(* IEC 61131-3 sources: TA/Tests/Diagnostic/Unitbus 0 (32) (part 2) *)

(* ---- UB_local_0_36_AIG16.st ---- *)
PROGRAM UB_local_0_36_AIG16

(***************************************************************************)
// НАСТРОЙКА ФБ
(***************************************************************************)

UB_0_32_AIG16_CH0_VAL_QUALITY_AD.Valid_down := AD_VALID_DOWN;
UB_0_32_AIG16_CH0_VAL_QUALITY_AD.Valid_up := AD_VALID_UP;
UB_0_32_AIG16_CH0_VAL_QUALITY_AD.IN0 := AD_IN0;
UB_0_32_AIG16_CH0_VAL_QUALITY_AD.IN100 := AD_IN100;

UB_0_32_AIG16_CH4_VAL_QUALITY_AD.Valid_down := AD_VALID_DOWN;
UB_0_32_AIG16_CH4_VAL_QUALITY_AD.Valid_up := AD_VALID_UP;
UB_0_32_AIG16_CH4_VAL_QUALITY_AD.IN0 := AD_IN0;
UB_0_32_AIG16_CH4_VAL_QUALITY_AD.IN100 := AD_IN100;

UB_0_32_AIG16_CH8_VAL_QUALITY_AD.Valid_down := AD_VALID_DOWN;
UB_0_32_AIG16_CH8_VAL_QUALITY_AD.Valid_up := AD_VALID_UP;
UB_0_32_AIG16_CH8_VAL_QUALITY_AD.IN0 := AD_IN0;
UB_0_32_AIG16_CH8_VAL_QUALITY_AD.IN100 := AD_IN100;

UB_0_32_AIG16_CH12_VAL_QUALITY_AD.Valid_down := AD_VALID_DOWN;
UB_0_32_AIG16_CH12_VAL_QUALITY_AD.Valid_up := AD_VALID_UP;
UB_0_32_AIG16_CH12_VAL_QUALITY_AD.IN0 := AD_IN0;
UB_0_32_AIG16_CH12_VAL_QUALITY_AD.IN100 := AD_IN100;

(***************************************************************************)
// СБРОС ОШИБОК
(***************************************************************************)

IF UB_0_32_AIG16_KVIT
    THEN UB_0_32_AIG16_KVIT := FALSE;
END_IF;

(***************************************************************************)
// КАНАЛ 0
(***************************************************************************)

UB_0_32_AIG16_CH0_VAL_MEASUREMENT := _IO_I21_AIG16_0_VAL.Measurement;

//Отказ сигнала
IF INT14(ANY_TO_DINT(_IO_I21_AIG16_0_VAL.Quality))
    THEN UB_0_32_AIG16_CH0_VAL_QUALITY_FAULT := TRUE;
    ELSE UB_0_32_AIG16_CH0_VAL_QUALITY_FAULT := FALSE;
END_IF;

// Проверка на ошибку
IF _IO_I21_AIG16_0_VAL.Quality = 0
    THEN UB_0_32_AIG16_CH0_VAL_QUALITY_ERROR := TRUE;
    ELSE UB_0_32_AIG16_CH0_VAL_QUALITY_ERROR := FALSE;
END_IF;

(***************************************************************************)
// КАНАЛ 4
(***************************************************************************)

UB_0_32_AIG16_CH4_VAL_MEASUREMENT := _IO_I21_AIG16_4_VAL.Measurement;

//Отказ сигнала
IF INT14(ANY_TO_DINT(_IO_I21_AIG16_4_VAL.Quality))
    THEN UB_0_32_AIG16_CH4_VAL_QUALITY_FAULT := TRUE;
    ELSE UB_0_32_AIG16_CH4_VAL_QUALITY_FAULT := FALSE;
END_IF;

// Проверка на ошибку
IF _IO_I21_AIG16_4_VAL.Quality = 0
    THEN UB_0_32_AIG16_CH4_VAL_QUALITY_ERROR := TRUE;
    ELSE UB_0_32_AIG16_CH4_VAL_QUALITY_ERROR := FALSE;
END_IF;

(***************************************************************************)
// КАНАЛ 8
(***************************************************************************)

UB_0_32_AIG16_CH8_VAL_MEASUREMENT := _IO_I21_AIG16_8_VAL.Measurement;

//Отказ сигнала
IF INT14(ANY_TO_DINT(_IO_I21_AIG16_8_VAL.Quality))
    THEN UB_0_32_AIG16_CH8_VAL_QUALITY_FAULT := TRUE;
    ELSE UB_0_32_AIG16_CH8_VAL_QUALITY_FAULT := FALSE;
END_IF;

// Проверка на ошибку
IF _IO_I21_AIG16_8_VAL.Quality = 0
    THEN UB_0_32_AIG16_CH8_VAL_QUALITY_ERROR := TRUE;
    ELSE UB_0_32_AIG16_CH8_VAL_QUALITY_ERROR := FALSE;
END_IF;

(***************************************************************************)
// КАНАЛ 12
(***************************************************************************)

UB_0_32_AIG16_CH12_VAL_MEASUREMENT := _IO_I21_AIG16_12_VAL.Measurement;

//Отказ сигнала
IF INT14(ANY_TO_DINT(_IO_I21_AIG16_12_VAL.Quality))
    THEN UB_0_32_AIG16_CH12_VAL_QUALITY_FAULT := TRUE;
    ELSE UB_0_32_AIG16_CH12_VAL_QUALITY_FAULT := FALSE;
END_IF;

// Проверка на ошибку
IF _IO_I21_AIG16_12_VAL.Quality = 0
    THEN UB_0_32_AIG16_CH12_VAL_QUALITY_ERROR := TRUE;
    ELSE UB_0_32_AIG16_CH12_VAL_QUALITY_ERROR := FALSE;
END_IF;

(***************************************************************************)
// ИНТЕГРАЛЬНЫЕ ПОКАЗАТЕЛИ
(***************************************************************************)

// Интегральный показателшь VAL.Quality
IF NOT INT0(UB_0_32_AIG16_CH0_VAL_QUALITY) AND
    NOT INT0(UB_0_32_AIG16_CH4_VAL_QUALITY) AND
    NOT INT0(UB_0_32_AIG16_CH8_VAL_QUALITY) AND
    NOT INT0(UB_0_32_AIG16_CH12_VAL_QUALITY)

    THEN UB_0_32_AIG16_INTEGRAL_VAL_QUALITY := TRUE;
    ELSE UB_0_32_AIG16_INTEGRAL_VAL_QUALITY := FALSE;
END_IF;

(***************************************************************************)
// ДИАГНОСТИКА ШИНЫ
(***************************************************************************)

// Диагностика 1 группы
// Адресное пространство не было найдено в Ubusdb
IF
    // Канал 0
    NOT INT4(ANY_TO_DINT(_IO_I21_AIG16_0_VAL.Quality)) AND
    NOT INT5(ANY_TO_DINT(_IO_I21_AIG16_0_VAL.Quality)) AND
    NOT INT6(ANY_TO_DINT(_IO_I21_AIG16_0_VAL.Quality)) AND
    NOT INT7(ANY_TO_DINT(_IO_I21_AIG16_0_VAL.Quality)) AND

    // Канал 1
    NOT INT4(ANY_TO_DINT(_IO_I21_AIG16_1_VAL.Quality)) AND
    NOT INT5(ANY_TO_DINT(_IO_I21_AIG16_1_VAL.Quality)) AND
    NOT INT6(ANY_TO_DINT(_IO_I21_AIG16_1_VAL.Quality)) AND
    NOT INT7(ANY_TO_DINT(_IO_I21_AIG16_1_VAL.Quality)) AND

    // Канал 2
    NOT INT4(ANY_TO_DINT(_IO_I21_AIG16_2_VAL.Quality)) AND
    NOT INT5(ANY_TO_DINT(_IO_I21_AIG16_2_VAL.Quality)) AND
    NOT INT6(ANY_TO_DINT(_IO_I21_AIG16_2_VAL.Quality)) AND
    NOT INT7(ANY_TO_DINT(_IO_I21_AIG16_2_VAL.Quality)) AND

    // Канал 3
    NOT INT4(ANY_TO_DINT(_IO_I21_AIG16_3_VAL.Quality)) AND
    NOT INT5(ANY_TO_DINT(_IO_I21_AIG16_3_VAL.Quality)) AND
    NOT INT6(ANY_TO_DINT(_IO_I21_AIG16_3_VAL.Quality)) AND
    NOT INT7(ANY_TO_DINT(_IO_I21_AIG16_3_VAL.Quality))

    THEN UB_0_32_AIG16_UNITBUS_VAL_QUALITY_GROUP_1 := 0;
END_IF;

// Не сошлась контрольная сумма данных
IF
    // Канал 0
    INT4(ANY_TO_DINT(_IO_I21_AIG16_0_VAL.Quality)) AND
    NOT INT5(ANY_TO_DINT(_IO_I21_AIG16_0_VAL.Quality)) AND
    NOT INT6(ANY_TO_DINT(_IO_I21_AIG16_0_VAL.Quality)) AND
    NOT INT7(ANY_TO_DINT(_IO_I21_AIG16_0_VAL.Quality)) AND

    // Канал 1
    INT4(ANY_TO_DINT(_IO_I21_AIG16_1_VAL.Quality)) AND
    NOT INT5(ANY_TO_DINT(_IO_I21_AIG16_1_VAL.Quality)) AND
    NOT INT6(ANY_TO_DINT(_IO_I21_AIG16_1_VAL.Quality)) AND
    NOT INT7(ANY_TO_DINT(_IO_I21_AIG16_1_VAL.Quality)) AND

    // Канал 2
    INT4(ANY_TO_DINT(_IO_I21_AIG16_2_VAL.Quality)) AND
    NOT INT5(ANY_TO_DINT(_IO_I21_AIG16_2_VAL.Quality)) AND
    NOT INT6(ANY_TO_DINT(_IO_I21_AIG16_2_VAL.Quality)) AND
    NOT INT7(ANY_TO_DINT(_IO_I21_AIG16_2_VAL.Quality)) AND

    // Канал 3
    INT4(ANY_TO_DINT(_IO_I21_AIG16_3_VAL.Quality)) AND
    NOT INT5(ANY_TO_DINT(_IO_I21_AIG16_3_VAL.Quality)) AND
    NOT INT6(ANY_TO_DINT(_IO_I21_AIG16_3_VAL.Quality)) AND
    NOT INT7(ANY_TO_DINT(_IO_I21_AIG16_3_VAL.Quality))

    THEN UB_0_32_AIG16_UNITBUS_VAL_QUALITY_GROUP_1 := 1;
END_IF;

// Не выставлены биты достоверности элементов в АП
IF
    // Канал 0
    NOT INT4(ANY_TO_DINT(_IO_I21_AIG16_0_VAL.Quality)) AND
    INT5(ANY_TO_DINT(_IO_I21_AIG16_0_VAL.Quality)) AND
    NOT INT6(ANY_TO_DINT(_IO_I21_AIG16_0_VAL.Quality)) AND
    NOT INT7(ANY_TO_DINT(_IO_I21_AIG16_0_VAL.Quality)) AND

    // Канал 1
    NOT INT4(ANY_TO_DINT(_IO_I21_AIG16_1_VAL.Quality)) AND
    INT5(ANY_TO_DINT(_IO_I21_AIG16_1_VAL.Quality)) AND
    NOT INT6(ANY_TO_DINT(_IO_I21_AIG16_1_VAL.Quality)) AND
    NOT INT7(ANY_TO_DINT(_IO_I21_AIG16_1_VAL.Quality)) AND

    // Канал 2
    NOT INT4(ANY_TO_DINT(_IO_I21_AIG16_2_VAL.Quality)) AND
    INT5(ANY_TO_DINT(_IO_I21_AIG16_2_VAL.Quality)) AND
    NOT INT6(ANY_TO_DINT(_IO_I21_AIG16_2_VAL.Quality)) AND
    NOT INT7(ANY_TO_DINT(_IO_I21_AIG16_2_VAL.Quality)) AND

    // Канал 3
    NOT INT4(ANY_TO_DINT(_IO_I21_AIG16_3_VAL.Quality)) AND
    INT5(ANY_TO_DINT(_IO_I21_AIG16_3_VAL.Quality)) AND
    NOT INT6(ANY_TO_DINT(_IO_I21_AIG16_3_VAL.Quality)) AND
    NOT INT7(ANY_TO_DINT(_IO_I21_AIG16_3_VAL.Quality))

    THEN UB_0_32_AIG16_UNITBUS_VAL_QUALITY_GROUP_1 := 2;
END_IF;

// Полученные данные корректны
IF
    // Канал 0
    INT4(ANY_TO_DINT(_IO_I21_AIG16_0_VAL.Quality)) AND
    INT5(ANY_TO_DINT(_IO_I21_AIG16_0_VAL.Quality)) AND
    NOT INT6(ANY_TO_DINT(_IO_I21_AIG16_0_VAL.Quality)) AND
    NOT INT7(ANY_TO_DINT(_IO_I21_AIG16_0_VAL.Quality)) AND

    // Канал 1
    INT4(ANY_TO_DINT(_IO_I21_AIG16_1_VAL.Quality)) AND
    INT5(ANY_TO_DINT(_IO_I21_AIG16_1_VAL.Quality)) AND
    NOT INT6(ANY_TO_DINT(_IO_I21_AIG16_1_VAL.Quality)) AND
    NOT INT7(ANY_TO_DINT(_IO_I21_AIG16_1_VAL.Quality)) AND

    // Канал 2
    INT4(ANY_TO_DINT(_IO_I21_AIG16_2_VAL.Quality)) AND
    INT5(ANY_TO_DINT(_IO_I21_AIG16_2_VAL.Quality)) AND
    NOT INT6(ANY_TO_DINT(_IO_I21_AIG16_2_VAL.Quality)) AND
    NOT INT7(ANY_TO_DINT(_IO_I21_AIG16_2_VAL.Quality)) AND

    // Канал 3
    INT4(ANY_TO_DINT(_IO_I21_AIG16_3_VAL.Quality)) AND
    INT5(ANY_TO_DINT(_IO_I21_AIG16_3_VAL.Quality)) AND
    NOT INT6(ANY_TO_DINT(_IO_I21_AIG16_3_VAL.Quality)) AND
    NOT INT7(ANY_TO_DINT(_IO_I21_AIG16_3_VAL.Quality))

    THEN UB_0_32_AIG16_UNITBUS_VAL_QUALITY_GROUP_1 := 3;
END_IF;

// Диагностика 2 группы
// Адресное пространство не было найдено в Ubusdb
IF
    // Канал 4
    NOT INT4(ANY_TO_DINT(_IO_I21_AIG16_4_VAL.Quality)) AND
    NOT INT5(ANY_TO_DINT(_IO_I21_AIG16_4_VAL.Quality)) AND
    NOT INT6(ANY_TO_DINT(_IO_I21_AIG16_4_VAL.Quality)) AND
    NOT INT7(ANY_TO_DINT(_IO_I21_AIG16_4_VAL.Quality)) AND

    // Канал 5
    NOT INT4(ANY_TO_DINT(_IO_I21_AIG16_5_VAL.Quality)) AND
    NOT INT5(ANY_TO_DINT(_IO_I21_AIG16_5_VAL.Quality)) AND
    NOT INT6(ANY_TO_DINT(_IO_I21_AIG16_5_VAL.Quality)) AND
    NOT INT7(ANY_TO_DINT(_IO_I21_AIG16_5_VAL.Quality)) AND

    // Канал 6
    NOT INT4(ANY_TO_DINT(_IO_I21_AIG16_6_VAL.Quality)) AND
    NOT INT5(ANY_TO_DINT(_IO_I21_AIG16_6_VAL.Quality)) AND
    NOT INT6(ANY_TO_DINT(_IO_I21_AIG16_6_VAL.Quality)) AND
    NOT INT7(ANY_TO_DINT(_IO_I21_AIG16_6_VAL.Quality)) AND

    // Канал 7
    NOT INT4(ANY_TO_DINT(_IO_I21_AIG16_7_VAL.Quality)) AND
    NOT INT5(ANY_TO_DINT(_IO_I21_AIG16_7_VAL.Quality)) AND
    NOT INT6(ANY_TO_DINT(_IO_I21_AIG16_7_VAL.Quality)) AND
    NOT INT7(ANY_TO_DINT(_IO_I21_AIG16_7_VAL.Quality))

    THEN UB_0_32_AIG16_UNITBUS_VAL_QUALITY_GROUP_2 := 0;
END_IF;

// Не сошлась контрольная сумма данных
IF
    // Канал 4
    INT4(ANY_TO_DINT(_IO_I21_AIG16_4_VAL.Quality)) AND
    NOT INT5(ANY_TO_DINT(_IO_I21_AIG16_4_VAL.Quality)) AND
    NOT INT6(ANY_TO_DINT(_IO_I21_AIG16_4_VAL.Quality)) AND
    NOT INT7(ANY_TO_DINT(_IO_I21_AIG16_4_VAL.Quality)) AND

    // Канал 5
    INT4(ANY_TO_DINT(_IO_I21_AIG16_5_VAL.Quality)) AND
    NOT INT5(ANY_TO_DINT(_IO_I21_AIG16_5_VAL.Quality)) AND
    NOT INT6(ANY_TO_DINT(_IO_I21_AIG16_5_VAL.Quality)) AND
    NOT INT7(ANY_TO_DINT(_IO_I21_AIG16_5_VAL.Quality)) AND

    // Канал 6
    INT4(ANY_TO_DINT(_IO_I21_AIG16_6_VAL.Quality)) AND
    NOT INT5(ANY_TO_DINT(_IO_I21_AIG16_6_VAL.Quality)) AND
    NOT INT6(ANY_TO_DINT(_IO_I21_AIG16_6_VAL.Quality)) AND
    NOT INT7(ANY_TO_DINT(_IO_I21_AIG16_6_VAL.Quality)) AND

    // Канал 7
    INT4(ANY_TO_DINT(_IO_I21_AIG16_7_VAL.Quality)) AND
    NOT INT5(ANY_TO_DINT(_IO_I21_AIG16_7_VAL.Quality)) AND
    NOT INT6(ANY_TO_DINT(_IO_I21_AIG16_7_VAL.Quality)) AND
    NOT INT7(ANY_TO_DINT(_IO_I21_AIG16_7_VAL.Quality))

    THEN UB_0_32_AIG16_UNITBUS_VAL_QUALITY_GROUP_2 := 1;
END_IF;

// Не выставлены биты достоверности элементов в АП
IF
    // Канал 4
    NOT INT4(ANY_TO_DINT(_IO_I21_AIG16_4_VAL.Quality)) AND
    INT5(ANY_TO_DINT(_IO_I21_AIG16_4_VAL.Quality)) AND
    NOT INT6(ANY_TO_DINT(_IO_I21_AIG16_4_VAL.Quality)) AND
    NOT INT7(ANY_TO_DINT(_IO_I21_AIG16_4_VAL.Quality)) AND

    // Канал 5
    NOT INT4(ANY_TO_DINT(_IO_I21_AIG16_5_VAL.Quality)) AND
    INT5(ANY_TO_DINT(_IO_I21_AIG16_5_VAL.Quality)) AND
    NOT INT6(ANY_TO_DINT(_IO_I21_AIG16_5_VAL.Quality)) AND
    NOT INT7(ANY_TO_DINT(_IO_I21_AIG16_5_VAL.Quality)) AND

    // Канал 6
    NOT INT4(ANY_TO_DINT(_IO_I21_AIG16_6_VAL.Quality)) AND
    INT5(ANY_TO_DINT(_IO_I21_AIG16_6_VAL.Quality)) AND
    NOT INT6(ANY_TO_DINT(_IO_I21_AIG16_6_VAL.Quality)) AND
    NOT INT7(ANY_TO_DINT(_IO_I21_AIG16_6_VAL.Quality)) AND

    // Канал 7
    NOT INT4(ANY_TO_DINT(_IO_I21_AIG16_7_VAL.Quality)) AND
    INT5(ANY_TO_DINT(_IO_I21_AIG16_7_VAL.Quality)) AND
    NOT INT6(ANY_TO_DINT(_IO_I21_AIG16_7_VAL.Quality)) AND
    NOT INT7(ANY_TO_DINT(_IO_I21_AIG16_7_VAL.Quality))

    THEN UB_0_32_AIG16_UNITBUS_VAL_QUALITY_GROUP_2 := 2;
END_IF;

// Полученные данные корректны
IF
    // Канал 4
    INT4(ANY_TO_DINT(_IO_I21_AIG16_4_VAL.Quality)) AND
    INT5(ANY_TO_DINT(_IO_I21_AIG16_4_VAL.Quality)) AND
    NOT INT6(ANY_TO_DINT(_IO_I21_AIG16_4_VAL.Quality)) AND
    NOT INT7(ANY_TO_DINT(_IO_I21_AIG16_4_VAL.Quality)) AND

    // Канал 5
    INT4(ANY_TO_DINT(_IO_I21_AIG16_5_VAL.Quality)) AND
    INT5(ANY_TO_DINT(_IO_I21_AIG16_5_VAL.Quality)) AND
    NOT INT6(ANY_TO_DINT(_IO_I21_AIG16_5_VAL.Quality)) AND
    NOT INT7(ANY_TO_DINT(_IO_I21_AIG16_5_VAL.Quality)) AND

    // Канал 6
    INT4(ANY_TO_DINT(_IO_I21_AIG16_6_VAL.Quality)) AND
    INT5(ANY_TO_DINT(_IO_I21_AIG16_6_VAL.Quality)) AND
    NOT INT6(ANY_TO_DINT(_IO_I21_AIG16_6_VAL.Quality)) AND
    NOT INT7(ANY_TO_DINT(_IO_I21_AIG16_6_VAL.Quality)) AND

    // Канал 7
    INT4(ANY_TO_DINT(_IO_I21_AIG16_7_VAL.Quality)) AND
    INT5(ANY_TO_DINT(_IO_I21_AIG16_7_VAL.Quality)) AND
    NOT INT6(ANY_TO_DINT(_IO_I21_AIG16_7_VAL.Quality)) AND
    NOT INT7(ANY_TO_DINT(_IO_I21_AIG16_7_VAL.Quality))

    THEN UB_0_32_AIG16_UNITBUS_VAL_QUALITY_GROUP_2 := 3;
END_IF;

// Диагностика 3 группы
// Адресное пространство не было найдено в Ubusdb
IF
    // Канал 8
    NOT INT4(ANY_TO_DINT(_IO_I21_AIG16_4_VAL.Quality)) AND
    NOT INT5(ANY_TO_DINT(_IO_I21_AIG16_4_VAL.Quality)) AND
    NOT INT6(ANY_TO_DINT(_IO_I21_AIG16_4_VAL.Quality)) AND
    NOT INT7(ANY_TO_DINT(_IO_I21_AIG16_4_VAL.Quality)) AND

    // Канал 9
    NOT INT4(ANY_TO_DINT(_IO_I21_AIG16_5_VAL.Quality)) AND
    NOT INT5(ANY_TO_DINT(_IO_I21_AIG16_5_VAL.Quality)) AND
    NOT INT6(ANY_TO_DINT(_IO_I21_AIG16_5_VAL.Quality)) AND
    NOT INT7(ANY_TO_DINT(_IO_I21_AIG16_5_VAL.Quality)) AND

    // Канал 10
    NOT INT4(ANY_TO_DINT(_IO_I21_AIG16_6_VAL.Quality)) AND
    NOT INT5(ANY_TO_DINT(_IO_I21_AIG16_6_VAL.Quality)) AND
    NOT INT6(ANY_TO_DINT(_IO_I21_AIG16_6_VAL.Quality)) AND
    NOT INT7(ANY_TO_DINT(_IO_I21_AIG16_6_VAL.Quality)) AND

    // Канал 11
    NOT INT4(ANY_TO_DINT(_IO_I21_AIG16_7_VAL.Quality)) AND
    NOT INT5(ANY_TO_DINT(_IO_I21_AIG16_7_VAL.Quality)) AND
    NOT INT6(ANY_TO_DINT(_IO_I21_AIG16_7_VAL.Quality)) AND
    NOT INT7(ANY_TO_DINT(_IO_I21_AIG16_7_VAL.Quality))

    THEN UB_0_32_AIG16_UNITBUS_VAL_QUALITY_GROUP_3 := 0;
END_IF;

// Не сошлась контрольная сумма данных
IF
    // Канал 8
    INT4(ANY_TO_DINT(_IO_I21_AIG16_4_VAL.Quality)) AND
    NOT INT5(ANY_TO_DINT(_IO_I21_AIG16_4_VAL.Quality)) AND
    NOT INT6(ANY_TO_DINT(_IO_I21_AIG16_4_VAL.Quality)) AND
    NOT INT7(ANY_TO_DINT(_IO_I21_AIG16_4_VAL.Quality)) AND

    // Канал 9
    INT4(ANY_TO_DINT(_IO_I21_AIG16_5_VAL.Quality)) AND
    NOT INT5(ANY_TO_DINT(_IO_I21_AIG16_5_VAL.Quality)) AND
    NOT INT6(ANY_TO_DINT(_IO_I21_AIG16_5_VAL.Quality)) AND
    NOT INT7(ANY_TO_DINT(_IO_I21_AIG16_5_VAL.Quality)) AND

    // Канал 10
    INT4(ANY_TO_DINT(_IO_I21_AIG16_6_VAL.Quality)) AND
    NOT INT5(ANY_TO_DINT(_IO_I21_AIG16_6_VAL.Quality)) AND
    NOT INT6(ANY_TO_DINT(_IO_I21_AIG16_6_VAL.Quality)) AND
    NOT INT7(ANY_TO_DINT(_IO_I21_AIG16_6_VAL.Quality)) AND

    // Канал 11
    INT4(ANY_TO_DINT(_IO_I21_AIG16_7_VAL.Quality)) AND
    NOT INT5(ANY_TO_DINT(_IO_I21_AIG16_7_VAL.Quality)) AND
    NOT INT6(ANY_TO_DINT(_IO_I21_AIG16_7_VAL.Quality)) AND
    NOT INT7(ANY_TO_DINT(_IO_I21_AIG16_7_VAL.Quality))

    THEN UB_0_32_AIG16_UNITBUS_VAL_QUALITY_GROUP_3 := 1;
END_IF;

// Не выставлены биты достоверности элементов в АП
IF
    // Канал 8
    NOT INT4(ANY_TO_DINT(_IO_I21_AIG16_4_VAL.Quality)) AND
    INT5(ANY_TO_DINT(_IO_I21_AIG16_4_VAL.Quality)) AND
    NOT INT6(ANY_TO_DINT(_IO_I21_AIG16_4_VAL.Quality)) AND
    NOT INT7(ANY_TO_DINT(_IO_I21_AIG16_4_VAL.Quality)) AND

    // Канал 9
    NOT INT4(ANY_TO_DINT(_IO_I21_AIG16_5_VAL.Quality)) AND
    INT5(ANY_TO_DINT(_IO_I21_AIG16_5_VAL.Quality)) AND
    NOT INT6(ANY_TO_DINT(_IO_I21_AIG16_5_VAL.Quality)) AND
    NOT INT7(ANY_TO_DINT(_IO_I21_AIG16_5_VAL.Quality)) AND

    // Канал 10
    NOT INT4(ANY_TO_DINT(_IO_I21_AIG16_6_VAL.Quality)) AND
    INT5(ANY_TO_DINT(_IO_I21_AIG16_6_VAL.Quality)) AND
    NOT INT6(ANY_TO_DINT(_IO_I21_AIG16_6_VAL.Quality)) AND
    NOT INT7(ANY_TO_DINT(_IO_I21_AIG16_6_VAL.Quality)) AND

    // Канал 11
    NOT INT4(ANY_TO_DINT(_IO_I21_AIG16_7_VAL.Quality)) AND
    INT5(ANY_TO_DINT(_IO_I21_AIG16_7_VAL.Quality)) AND
    NOT INT6(ANY_TO_DINT(_IO_I21_AIG16_7_VAL.Quality)) AND
    NOT INT7(ANY_TO_DINT(_IO_I21_AIG16_7_VAL.Quality))

    THEN UB_0_32_AIG16_UNITBUS_VAL_QUALITY_GROUP_3 := 2;
END_IF;

// Полученные данные корректны
IF
    // Канал 8
    INT4(ANY_TO_DINT(_IO_I21_AIG16_4_VAL.Quality)) AND
    INT5(ANY_TO_DINT(_IO_I21_AIG16_4_VAL.Quality)) AND
    NOT INT6(ANY_TO_DINT(_IO_I21_AIG16_4_VAL.Quality)) AND
    NOT INT7(ANY_TO_DINT(_IO_I21_AIG16_4_VAL.Quality)) AND

    // Канал 9
    INT4(ANY_TO_DINT(_IO_I21_AIG16_5_VAL.Quality)) AND
    INT5(ANY_TO_DINT(_IO_I21_AIG16_5_VAL.Quality)) AND
    NOT INT6(ANY_TO_DINT(_IO_I21_AIG16_5_VAL.Quality)) AND
    NOT INT7(ANY_TO_DINT(_IO_I21_AIG16_5_VAL.Quality)) AND

    // Канал 10
    INT4(ANY_TO_DINT(_IO_I21_AIG16_6_VAL.Quality)) AND
    INT5(ANY_TO_DINT(_IO_I21_AIG16_6_VAL.Quality)) AND
    NOT INT6(ANY_TO_DINT(_IO_I21_AIG16_6_VAL.Quality)) AND
    NOT INT7(ANY_TO_DINT(_IO_I21_AIG16_6_VAL.Quality)) AND

    // Канал 11
    INT4(ANY_TO_DINT(_IO_I21_AIG16_7_VAL.Quality)) AND
    INT5(ANY_TO_DINT(_IO_I21_AIG16_7_VAL.Quality)) AND
    NOT INT6(ANY_TO_DINT(_IO_I21_AIG16_7_VAL.Quality)) AND
    NOT INT7(ANY_TO_DINT(_IO_I21_AIG16_7_VAL.Quality))

    THEN UB_0_32_AIG16_UNITBUS_VAL_QUALITY_GROUP_3 := 3;
END_IF;

// Диагностика 4 группы
// Адресное пространство не было найдено в Ubusdb
IF
    // Канал 12
    NOT INT4(ANY_TO_DINT(_IO_I21_AIG16_12_VAL.Quality)) AND
    NOT INT5(ANY_TO_DINT(_IO_I21_AIG16_12_VAL.Quality)) AND
    NOT INT6(ANY_TO_DINT(_IO_I21_AIG16_12_VAL.Quality)) AND
    NOT INT7(ANY_TO_DINT(_IO_I21_AIG16_12_VAL.Quality)) AND

    // Канал 13
    NOT INT4(ANY_TO_DINT(_IO_I21_AIG16_13_VAL.Quality)) AND
    NOT INT5(ANY_TO_DINT(_IO_I21_AIG16_13_VAL.Quality)) AND
    NOT INT6(ANY_TO_DINT(_IO_I21_AIG16_13_VAL.Quality)) AND
    NOT INT7(ANY_TO_DINT(_IO_I21_AIG16_13_VAL.Quality)) AND

    // Канал 14
    NOT INT4(ANY_TO_DINT(_IO_I21_AIG16_14_VAL.Quality)) AND
    NOT INT5(ANY_TO_DINT(_IO_I21_AIG16_14_VAL.Quality)) AND
    NOT INT6(ANY_TO_DINT(_IO_I21_AIG16_14_VAL.Quality)) AND
    NOT INT7(ANY_TO_DINT(_IO_I21_AIG16_14_VAL.Quality)) AND

    // Канал 15
    NOT INT4(ANY_TO_DINT(_IO_I21_AIG16_15_VAL.Quality)) AND
    NOT INT5(ANY_TO_DINT(_IO_I21_AIG16_15_VAL.Quality)) AND
    NOT INT6(ANY_TO_DINT(_IO_I21_AIG16_15_VAL.Quality)) AND
    NOT INT7(ANY_TO_DINT(_IO_I21_AIG16_15_VAL.Quality))

    THEN UB_0_32_AIG16_UNITBUS_VAL_QUALITY_GROUP_4 := 0;
END_IF;

// Не сошлась контрольная сумма данных
IF
    // Канал 12
    INT4(ANY_TO_DINT(_IO_I21_AIG16_12_VAL.Quality)) AND
    NOT INT5(ANY_TO_DINT(_IO_I21_AIG16_12_VAL.Quality)) AND
    NOT INT6(ANY_TO_DINT(_IO_I21_AIG16_12_VAL.Quality)) AND
    NOT INT7(ANY_TO_DINT(_IO_I21_AIG16_12_VAL.Quality)) AND

    // Канал 13
    INT4(ANY_TO_DINT(_IO_I21_AIG16_13_VAL.Quality)) AND
    NOT INT5(ANY_TO_DINT(_IO_I21_AIG16_13_VAL.Quality)) AND
    NOT INT6(ANY_TO_DINT(_IO_I21_AIG16_13_VAL.Quality)) AND
    NOT INT7(ANY_TO_DINT(_IO_I21_AIG16_13_VAL.Quality)) AND

    // Канал 14
    INT4(ANY_TO_DINT(_IO_I21_AIG16_14_VAL.Quality)) AND
    NOT INT5(ANY_TO_DINT(_IO_I21_AIG16_14_VAL.Quality)) AND
    NOT INT6(ANY_TO_DINT(_IO_I21_AIG16_14_VAL.Quality)) AND
    NOT INT7(ANY_TO_DINT(_IO_I21_AIG16_14_VAL.Quality)) AND

    // Канал 15
    INT4(ANY_TO_DINT(_IO_I21_AIG16_15_VAL.Quality)) AND
    NOT INT5(ANY_TO_DINT(_IO_I21_AIG16_15_VAL.Quality)) AND
    NOT INT6(ANY_TO_DINT(_IO_I21_AIG16_15_VAL.Quality)) AND
    NOT INT7(ANY_TO_DINT(_IO_I21_AIG16_15_VAL.Quality))

    THEN UB_0_32_AIG16_UNITBUS_VAL_QUALITY_GROUP_4 := 1;
END_IF;

// Не выставлены биты достоверности элементов в АП
IF
    // Канал 12
    NOT INT4(ANY_TO_DINT(_IO_I21_AIG16_12_VAL.Quality)) AND
    INT5(ANY_TO_DINT(_IO_I21_AIG16_12_VAL.Quality)) AND
    NOT INT6(ANY_TO_DINT(_IO_I21_AIG16_12_VAL.Quality)) AND
    NOT INT7(ANY_TO_DINT(_IO_I21_AIG16_12_VAL.Quality)) AND

    // Канал 13
    NOT INT4(ANY_TO_DINT(_IO_I21_AIG16_13_VAL.Quality)) AND
    INT5(ANY_TO_DINT(_IO_I21_AIG16_13_VAL.Quality)) AND
    NOT INT6(ANY_TO_DINT(_IO_I21_AIG16_13_VAL.Quality)) AND
    NOT INT7(ANY_TO_DINT(_IO_I21_AIG16_13_VAL.Quality)) AND

    // Канал 14
    NOT INT4(ANY_TO_DINT(_IO_I21_AIG16_14_VAL.Quality)) AND
    INT5(ANY_TO_DINT(_IO_I21_AIG16_14_VAL.Quality)) AND
    NOT INT6(ANY_TO_DINT(_IO_I21_AIG16_14_VAL.Quality)) AND
    NOT INT7(ANY_TO_DINT(_IO_I21_AIG16_14_VAL.Quality)) AND

    // Канал 15
    NOT INT4(ANY_TO_DINT(_IO_I21_AIG16_15_VAL.Quality)) AND
    INT5(ANY_TO_DINT(_IO_I21_AIG16_15_VAL.Quality)) AND
    NOT INT6(ANY_TO_DINT(_IO_I21_AIG16_15_VAL.Quality)) AND
    NOT INT7(ANY_TO_DINT(_IO_I21_AIG16_15_VAL.Quality))

    THEN UB_0_32_AIG16_UNITBUS_VAL_QUALITY_GROUP_4 := 2;
END_IF;

// Полученные данные корректны
IF
    // Канал 12
    INT4(ANY_TO_DINT(_IO_I21_AIG16_12_VAL.Quality)) AND
    INT5(ANY_TO_DINT(_IO_I21_AIG16_12_VAL.Quality)) AND
    NOT INT6(ANY_TO_DINT(_IO_I21_AIG16_12_VAL.Quality)) AND
    NOT INT7(ANY_TO_DINT(_IO_I21_AIG16_12_VAL.Quality)) AND

    // Канал 13
    INT4(ANY_TO_DINT(_IO_I21_AIG16_13_VAL.Quality)) AND
    INT5(ANY_TO_DINT(_IO_I21_AIG16_13_VAL.Quality)) AND
    NOT INT6(ANY_TO_DINT(_IO_I21_AIG16_13_VAL.Quality)) AND
    NOT INT7(ANY_TO_DINT(_IO_I21_AIG16_13_VAL.Quality)) AND

    // Канал 14
    INT4(ANY_TO_DINT(_IO_I21_AIG16_14_VAL.Quality)) AND
    INT5(ANY_TO_DINT(_IO_I21_AIG16_14_VAL.Quality)) AND
    NOT INT6(ANY_TO_DINT(_IO_I21_AIG16_14_VAL.Quality)) AND
    NOT INT7(ANY_TO_DINT(_IO_I21_AIG16_14_VAL.Quality)) AND

    // Канал 15
    INT4(ANY_TO_DINT(_IO_I21_AIG16_15_VAL.Quality)) AND
    INT5(ANY_TO_DINT(_IO_I21_AIG16_15_VAL.Quality)) AND
    NOT INT6(ANY_TO_DINT(_IO_I21_AIG16_15_VAL.Quality)) AND
    NOT INT7(ANY_TO_DINT(_IO_I21_AIG16_15_VAL.Quality))

    THEN UB_0_32_AIG16_UNITBUS_VAL_QUALITY_GROUP_4 := 3;
END_IF;

(***************************************************************************)
// ОБЩИЙ ИНТЕГРАЛЬНЫЙ ПОАЗАТЕЛЬ
(***************************************************************************)

// Адресное пространство не было найдено в Ubusdb
IF UB_0_32_AIG16_UNITBUS_VAL_QUALITY_GROUP_1 = 0 AND
    UB_0_32_AIG16_UNITBUS_VAL_QUALITY_GROUP_2 = 0 AND
    UB_0_32_AIG16_UNITBUS_VAL_QUALITY_GROUP_3 = 0 AND
    UB_0_32_AIG16_UNITBUS_VAL_QUALITY_GROUP_4 = 0

    THEN UB_0_32_AIG16_UNITBUS_VAL_QUALITY := 0;
END_IF;

// Не сошлась контрольная сумма данных
IF UB_0_32_AIG16_UNITBUS_VAL_QUALITY_GROUP_1 = 1 AND
    UB_0_32_AIG16_UNITBUS_VAL_QUALITY_GROUP_2 = 1 AND
    UB_0_32_AIG16_UNITBUS_VAL_QUALITY_GROUP_3 = 1 AND
    UB_0_32_AIG16_UNITBUS_VAL_QUALITY_GROUP_4 = 1

    THEN UB_0_32_AIG16_UNITBUS_VAL_QUALITY := 1;
END_IF;

// Не выставлены биты достоверности элементов в АП
IF UB_0_32_AIG16_UNITBUS_VAL_QUALITY_GROUP_1 = 2 AND
    UB_0_32_AIG16_UNITBUS_VAL_QUALITY_GROUP_2 = 2 AND
    UB_0_32_AIG16_UNITBUS_VAL_QUALITY_GROUP_3 = 2 AND
    UB_0_32_AIG16_UNITBUS_VAL_QUALITY_GROUP_4 = 2

    THEN UB_0_32_AIG16_UNITBUS_VAL_QUALITY := 2;
END_IF;

// Полученные данные корректны
IF UB_0_32_AIG16_UNITBUS_VAL_QUALITY_GROUP_1 = 3 AND
    UB_0_32_AIG16_UNITBUS_VAL_QUALITY_GROUP_2 = 3 AND
    UB_0_32_AIG16_UNITBUS_VAL_QUALITY_GROUP_3 = 3 AND
    UB_0_32_AIG16_UNITBUS_VAL_QUALITY_GROUP_4 = 3

    THEN UB_0_32_AIG16_UNITBUS_VAL_QUALITY := 3;
END_IF;

END_PROGRAM

(* ---- UB_local_0_37_AI8.st ---- *)
PROGRAM UB_local_0_37_AI8

(***************************************************************************)
// НАСТРОЙКА ФБ
(***************************************************************************)

UB_0_32_AI8_CH0_VAL_QUALITY_AD.Valid_down := AD_VALID_DOWN;
UB_0_32_AI8_CH0_VAL_QUALITY_AD.Valid_up := AD_VALID_UP;
UB_0_32_AI8_CH0_VAL_QUALITY_AD.IN0 := AD_IN0;
UB_0_32_AI8_CH0_VAL_QUALITY_AD.IN100 := AD_IN100;

UB_0_32_AI8_CH4_VAL_QUALITY_AD.Valid_down := AD_VALID_DOWN;
UB_0_32_AI8_CH4_VAL_QUALITY_AD.Valid_up := AD_VALID_UP;
UB_0_32_AI8_CH4_VAL_QUALITY_AD.IN0 := AD_IN0;
UB_0_32_AI8_CH4_VAL_QUALITY_AD.IN100 := AD_IN100;

(***************************************************************************)
// СБРОС ОШИБОК
(***************************************************************************)

IF UB_0_32_AI8_KVIT
    THEN UB_0_32_AI8_KVIT := FALSE;
END_IF;

(***************************************************************************)
// КАНАЛ 0
(***************************************************************************)

UB_0_32_AI8_CH0_VAL_MEASUREMENT := _IO_I22_AI8_0_VAL.Measurement;

//Отказ сигнала
IF INT14(ANY_TO_DINT(_IO_I22_AI8_0_VAL.Quality))
    THEN UB_0_32_AI8_CH0_VAL_QUALITY_FAULT := TRUE;
    ELSE UB_0_32_AI8_CH0_VAL_QUALITY_FAULT := FALSE;
END_IF;

// Проверка на ошибку
IF _IO_I22_AI8_0_VAL.Quality = 0
    THEN UB_0_32_AI8_CH0_VAL_QUALITY_ERROR := TRUE;
    ELSE UB_0_32_AI8_CH0_VAL_QUALITY_ERROR := FALSE;
END_IF;

(***************************************************************************)
// КАНАЛ 4
(***************************************************************************)

UB_0_32_AI8_CH4_VAL_MEASUREMENT := _IO_I22_AI8_4_VAL.Measurement;

//Отказ сигнала
IF INT14(ANY_TO_DINT(_IO_I22_AI8_4_VAL.Quality))
    THEN UB_0_32_AI8_CH4_VAL_QUALITY_FAULT := TRUE;
    ELSE UB_0_32_AI8_CH4_VAL_QUALITY_FAULT := FALSE;
END_IF;

// Проверка на ошибку
IF _IO_I22_AI8_4_VAL.Quality = 0
    THEN UB_0_32_AI8_CH4_VAL_QUALITY_ERROR := TRUE;
    ELSE UB_0_32_AI8_CH4_VAL_QUALITY_ERROR := FALSE;
END_IF;

(***************************************************************************)
// ИНТЕГРАЛЬНЫЕ ПОКАЗАТЕЛИ
(***************************************************************************)

// Интегральный показателшь VAL.Quality
IF NOT INT0(UB_0_32_AI8_CH0_VAL_QUALITY) AND
    NOT INT0(UB_0_32_AI8_CH4_VAL_QUALITY)

    THEN UB_0_32_AI8_INTEGRAL_VAL_QUALITY := TRUE;
    ELSE UB_0_32_AI8_INTEGRAL_VAL_QUALITY := FALSE;
END_IF;

(***************************************************************************)
// ДИАГНОСТИКА ШИНЫ
(***************************************************************************)

// Диагностика 1 группы
// Адресное пространство не было найдено в Ubusdb
IF
    // Канал 0
    NOT INT4(ANY_TO_DINT(_IO_I22_AI8_0_VAL.Quality)) AND
    NOT INT5(ANY_TO_DINT(_IO_I22_AI8_0_VAL.Quality)) AND
    NOT INT6(ANY_TO_DINT(_IO_I22_AI8_0_VAL.Quality)) AND
    NOT INT7(ANY_TO_DINT(_IO_I22_AI8_0_VAL.Quality)) AND

    // Канал 1
    NOT INT4(ANY_TO_DINT(_IO_I22_AI8_1_VAL.Quality)) AND
    NOT INT5(ANY_TO_DINT(_IO_I22_AI8_1_VAL.Quality)) AND
    NOT INT6(ANY_TO_DINT(_IO_I22_AI8_1_VAL.Quality)) AND
    NOT INT7(ANY_TO_DINT(_IO_I22_AI8_1_VAL.Quality)) AND

    // Канал 2
    NOT INT4(ANY_TO_DINT(_IO_I22_AI8_2_VAL.Quality)) AND
    NOT INT5(ANY_TO_DINT(_IO_I22_AI8_2_VAL.Quality)) AND
    NOT INT6(ANY_TO_DINT(_IO_I22_AI8_2_VAL.Quality)) AND
    NOT INT7(ANY_TO_DINT(_IO_I22_AI8_2_VAL.Quality)) AND

    // Канал 3
    NOT INT4(ANY_TO_DINT(_IO_I22_AI8_3_VAL.Quality)) AND
    NOT INT5(ANY_TO_DINT(_IO_I22_AI8_3_VAL.Quality)) AND
    NOT INT6(ANY_TO_DINT(_IO_I22_AI8_3_VAL.Quality)) AND
    NOT INT7(ANY_TO_DINT(_IO_I22_AI8_3_VAL.Quality))

    THEN UB_0_32_AI8_UNITBUS_VAL_QUALITY_GROUP_1 := 0;
END_IF;

// Не сошлась контрольная сумма данных
IF
    // Канал 0
    INT4(ANY_TO_DINT(_IO_I22_AI8_0_VAL.Quality)) AND
    NOT INT5(ANY_TO_DINT(_IO_I22_AI8_0_VAL.Quality)) AND
    NOT INT6(ANY_TO_DINT(_IO_I22_AI8_0_VAL.Quality)) AND
    NOT INT7(ANY_TO_DINT(_IO_I22_AI8_0_VAL.Quality)) AND

    // Канал 1
    INT4(ANY_TO_DINT(_IO_I22_AI8_1_VAL.Quality)) AND
    NOT INT5(ANY_TO_DINT(_IO_I22_AI8_1_VAL.Quality)) AND
    NOT INT6(ANY_TO_DINT(_IO_I22_AI8_1_VAL.Quality)) AND
    NOT INT7(ANY_TO_DINT(_IO_I22_AI8_1_VAL.Quality)) AND

    // Канал 2
    INT4(ANY_TO_DINT(_IO_I22_AI8_2_VAL.Quality)) AND
    NOT INT5(ANY_TO_DINT(_IO_I22_AI8_2_VAL.Quality)) AND
    NOT INT6(ANY_TO_DINT(_IO_I22_AI8_2_VAL.Quality)) AND
    NOT INT7(ANY_TO_DINT(_IO_I22_AI8_2_VAL.Quality)) AND

    // Канал 3
    INT4(ANY_TO_DINT(_IO_I22_AI8_3_VAL.Quality)) AND
    NOT INT5(ANY_TO_DINT(_IO_I22_AI8_3_VAL.Quality)) AND
    NOT INT6(ANY_TO_DINT(_IO_I22_AI8_3_VAL.Quality)) AND
    NOT INT7(ANY_TO_DINT(_IO_I22_AI8_3_VAL.Quality))

    THEN UB_0_32_AI8_UNITBUS_VAL_QUALITY_GROUP_1 := 1;
END_IF;

// Не выставлены биты достоверности элементов в АП
IF
    // Канал 0
    NOT INT4(ANY_TO_DINT(_IO_I22_AI8_0_VAL.Quality)) AND
    INT5(ANY_TO_DINT(_IO_I22_AI8_0_VAL.Quality)) AND
    NOT INT6(ANY_TO_DINT(_IO_I22_AI8_0_VAL.Quality)) AND
    NOT INT7(ANY_TO_DINT(_IO_I22_AI8_0_VAL.Quality)) AND

    // Канал 1
    NOT INT4(ANY_TO_DINT(_IO_I22_AI8_1_VAL.Quality)) AND
    INT5(ANY_TO_DINT(_IO_I22_AI8_1_VAL.Quality)) AND
    NOT INT6(ANY_TO_DINT(_IO_I22_AI8_1_VAL.Quality)) AND
    NOT INT7(ANY_TO_DINT(_IO_I22_AI8_1_VAL.Quality)) AND

    // Канал 2
    NOT INT4(ANY_TO_DINT(_IO_I22_AI8_2_VAL.Quality)) AND
    INT5(ANY_TO_DINT(_IO_I22_AI8_2_VAL.Quality)) AND
    NOT INT6(ANY_TO_DINT(_IO_I22_AI8_2_VAL.Quality)) AND
    NOT INT7(ANY_TO_DINT(_IO_I22_AI8_2_VAL.Quality)) AND

    // Канал 3
    NOT INT4(ANY_TO_DINT(_IO_I22_AI8_3_VAL.Quality)) AND
    INT5(ANY_TO_DINT(_IO_I22_AI8_3_VAL.Quality)) AND
    NOT INT6(ANY_TO_DINT(_IO_I22_AI8_3_VAL.Quality)) AND
    NOT INT7(ANY_TO_DINT(_IO_I22_AI8_3_VAL.Quality))

    THEN UB_0_32_AI8_UNITBUS_VAL_QUALITY_GROUP_1 := 2;
END_IF;

// Полученные данные корректны
IF
    // Канал 0
    INT4(ANY_TO_DINT(_IO_I22_AI8_0_VAL.Quality)) AND
    INT5(ANY_TO_DINT(_IO_I22_AI8_0_VAL.Quality)) AND
    NOT INT6(ANY_TO_DINT(_IO_I22_AI8_0_VAL.Quality)) AND
    NOT INT7(ANY_TO_DINT(_IO_I22_AI8_0_VAL.Quality)) AND

    // Канал 1
    INT4(ANY_TO_DINT(_IO_I22_AI8_1_VAL.Quality)) AND
    INT5(ANY_TO_DINT(_IO_I22_AI8_1_VAL.Quality)) AND
    NOT INT6(ANY_TO_DINT(_IO_I22_AI8_1_VAL.Quality)) AND
    NOT INT7(ANY_TO_DINT(_IO_I22_AI8_1_VAL.Quality)) AND

    // Канал 2
    INT4(ANY_TO_DINT(_IO_I22_AI8_2_VAL.Quality)) AND
    INT5(ANY_TO_DINT(_IO_I22_AI8_2_VAL.Quality)) AND
    NOT INT6(ANY_TO_DINT(_IO_I22_AI8_2_VAL.Quality)) AND
    NOT INT7(ANY_TO_DINT(_IO_I22_AI8_2_VAL.Quality)) AND

    // Канал 3
    INT4(ANY_TO_DINT(_IO_I22_AI8_3_VAL.Quality)) AND
    INT5(ANY_TO_DINT(_IO_I22_AI8_3_VAL.Quality)) AND
    NOT INT6(ANY_TO_DINT(_IO_I22_AI8_3_VAL.Quality)) AND
    NOT INT7(ANY_TO_DINT(_IO_I22_AI8_3_VAL.Quality))

    THEN UB_0_32_AI8_UNITBUS_VAL_QUALITY_GROUP_1 := 3;
END_IF;

// Диагностика 2 группы
// Адресное пространство не было найдено в Ubusdb
IF
    // Канал 4
    NOT INT4(ANY_TO_DINT(_IO_I22_AI8_4_VAL.Quality)) AND
    NOT INT5(ANY_TO_DINT(_IO_I22_AI8_4_VAL.Quality)) AND
    NOT INT6(ANY_TO_DINT(_IO_I22_AI8_4_VAL.Quality)) AND
    NOT INT7(ANY_TO_DINT(_IO_I22_AI8_4_VAL.Quality)) AND

    // Канал 5
    NOT INT4(ANY_TO_DINT(_IO_I22_AI8_5_VAL.Quality)) AND
    NOT INT5(ANY_TO_DINT(_IO_I22_AI8_5_VAL.Quality)) AND
    NOT INT6(ANY_TO_DINT(_IO_I22_AI8_5_VAL.Quality)) AND
    NOT INT7(ANY_TO_DINT(_IO_I22_AI8_5_VAL.Quality)) AND

    // Канал 6
    NOT INT4(ANY_TO_DINT(_IO_I22_AI8_6_VAL.Quality)) AND
    NOT INT5(ANY_TO_DINT(_IO_I22_AI8_6_VAL.Quality)) AND
    NOT INT6(ANY_TO_DINT(_IO_I22_AI8_6_VAL.Quality)) AND
    NOT INT7(ANY_TO_DINT(_IO_I22_AI8_6_VAL.Quality)) AND

    // Канал 7
    NOT INT4(ANY_TO_DINT(_IO_I22_AI8_7_VAL.Quality)) AND
    NOT INT5(ANY_TO_DINT(_IO_I22_AI8_7_VAL.Quality)) AND
    NOT INT6(ANY_TO_DINT(_IO_I22_AI8_7_VAL.Quality)) AND
    NOT INT7(ANY_TO_DINT(_IO_I22_AI8_7_VAL.Quality))

    THEN UB_0_32_AI8_UNITBUS_VAL_QUALITY_GROUP_2 := 0;
END_IF;

// Не сошлась контрольная сумма данных
IF
    // Канал 4
    INT4(ANY_TO_DINT(_IO_I22_AI8_4_VAL.Quality)) AND
    NOT INT5(ANY_TO_DINT(_IO_I22_AI8_4_VAL.Quality)) AND
    NOT INT6(ANY_TO_DINT(_IO_I22_AI8_4_VAL.Quality)) AND
    NOT INT7(ANY_TO_DINT(_IO_I22_AI8_4_VAL.Quality)) AND

    // Канал 5
    INT4(ANY_TO_DINT(_IO_I22_AI8_5_VAL.Quality)) AND
    NOT INT5(ANY_TO_DINT(_IO_I22_AI8_5_VAL.Quality)) AND
    NOT INT6(ANY_TO_DINT(_IO_I22_AI8_5_VAL.Quality)) AND
    NOT INT7(ANY_TO_DINT(_IO_I22_AI8_5_VAL.Quality)) AND

    // Канал 6
    INT4(ANY_TO_DINT(_IO_I22_AI8_6_VAL.Quality)) AND
    NOT INT5(ANY_TO_DINT(_IO_I22_AI8_6_VAL.Quality)) AND
    NOT INT6(ANY_TO_DINT(_IO_I22_AI8_6_VAL.Quality)) AND
    NOT INT7(ANY_TO_DINT(_IO_I22_AI8_6_VAL.Quality)) AND

    // Канал 7
    INT4(ANY_TO_DINT(_IO_I22_AI8_7_VAL.Quality)) AND
    NOT INT5(ANY_TO_DINT(_IO_I22_AI8_7_VAL.Quality)) AND
    NOT INT6(ANY_TO_DINT(_IO_I22_AI8_7_VAL.Quality)) AND
    NOT INT7(ANY_TO_DINT(_IO_I22_AI8_7_VAL.Quality))

    THEN UB_0_32_AI8_UNITBUS_VAL_QUALITY_GROUP_2 := 1;
END_IF;

// Не выставлены биты достоверности элементов в АП
IF
    // Канал 4
    NOT INT4(ANY_TO_DINT(_IO_I22_AI8_4_VAL.Quality)) AND
    INT5(ANY_TO_DINT(_IO_I22_AI8_4_VAL.Quality)) AND
    NOT INT6(ANY_TO_DINT(_IO_I22_AI8_4_VAL.Quality)) AND
    NOT INT7(ANY_TO_DINT(_IO_I22_AI8_4_VAL.Quality)) AND

    // Канал 5
    NOT INT4(ANY_TO_DINT(_IO_I22_AI8_5_VAL.Quality)) AND
    INT5(ANY_TO_DINT(_IO_I22_AI8_5_VAL.Quality)) AND
    NOT INT6(ANY_TO_DINT(_IO_I22_AI8_5_VAL.Quality)) AND
    NOT INT7(ANY_TO_DINT(_IO_I22_AI8_5_VAL.Quality)) AND

    // Канал 6
    NOT INT4(ANY_TO_DINT(_IO_I22_AI8_6_VAL.Quality)) AND
    INT5(ANY_TO_DINT(_IO_I22_AI8_6_VAL.Quality)) AND
    NOT INT6(ANY_TO_DINT(_IO_I22_AI8_6_VAL.Quality)) AND
    NOT INT7(ANY_TO_DINT(_IO_I22_AI8_6_VAL.Quality)) AND

    // Канал 7
    NOT INT4(ANY_TO_DINT(_IO_I22_AI8_7_VAL.Quality)) AND
    INT5(ANY_TO_DINT(_IO_I22_AI8_7_VAL.Quality)) AND
    NOT INT6(ANY_TO_DINT(_IO_I22_AI8_7_VAL.Quality)) AND
    NOT INT7(ANY_TO_DINT(_IO_I22_AI8_7_VAL.Quality))

    THEN UB_0_32_AI8_UNITBUS_VAL_QUALITY_GROUP_2 := 2;
END_IF;

// Полученные данные корректны
IF
    // Канал 4
    INT4(ANY_TO_DINT(_IO_I22_AI8_4_VAL.Quality)) AND
    INT5(ANY_TO_DINT(_IO_I22_AI8_4_VAL.Quality)) AND
    NOT INT6(ANY_TO_DINT(_IO_I22_AI8_4_VAL.Quality)) AND
    NOT INT7(ANY_TO_DINT(_IO_I22_AI8_4_VAL.Quality)) AND

    // Канал 5
    INT4(ANY_TO_DINT(_IO_I22_AI8_5_VAL.Quality)) AND
    INT5(ANY_TO_DINT(_IO_I22_AI8_5_VAL.Quality)) AND
    NOT INT6(ANY_TO_DINT(_IO_I22_AI8_5_VAL.Quality)) AND
    NOT INT7(ANY_TO_DINT(_IO_I22_AI8_5_VAL.Quality)) AND

    // Канал 6
    INT4(ANY_TO_DINT(_IO_I22_AI8_6_VAL.Quality)) AND
    INT5(ANY_TO_DINT(_IO_I22_AI8_6_VAL.Quality)) AND
    NOT INT6(ANY_TO_DINT(_IO_I22_AI8_6_VAL.Quality)) AND
    NOT INT7(ANY_TO_DINT(_IO_I22_AI8_6_VAL.Quality)) AND

    // Канал 7
    INT4(ANY_TO_DINT(_IO_I22_AI8_7_VAL.Quality)) AND
    INT5(ANY_TO_DINT(_IO_I22_AI8_7_VAL.Quality)) AND
    NOT INT6(ANY_TO_DINT(_IO_I22_AI8_7_VAL.Quality)) AND
    NOT INT7(ANY_TO_DINT(_IO_I22_AI8_7_VAL.Quality))

    THEN UB_0_32_AI8_UNITBUS_VAL_QUALITY_GROUP_2 := 3;
END_IF;

(***************************************************************************)
// ОБЩИЙ ИНТЕГРАЛЬНЫЙ ПОАЗАТЕЛЬ
(***************************************************************************)

// Адресное пространство не было найдено в Ubusdb
IF UB_0_32_AI8_UNITBUS_VAL_QUALITY_GROUP_1 = 0 AND
    UB_0_32_AI8_UNITBUS_VAL_QUALITY_GROUP_2 = 0

    THEN UB_0_32_AI8_UNITBUS_VAL_QUALITY := 0;
END_IF;

// Не сошлась контрольная сумма данных
IF UB_0_32_AI8_UNITBUS_VAL_QUALITY_GROUP_1 = 1 AND
    UB_0_32_AI8_UNITBUS_VAL_QUALITY_GROUP_2 = 1

    THEN UB_0_32_AI8_UNITBUS_VAL_QUALITY := 1;
END_IF;

// Не выставлены биты достоверности элементов в АП
IF UB_0_32_AI8_UNITBUS_VAL_QUALITY_GROUP_1 = 2 AND
    UB_0_32_AI8_UNITBUS_VAL_QUALITY_GROUP_2 = 2

    THEN UB_0_32_AI8_UNITBUS_VAL_QUALITY := 2;
END_IF;

// Полученные данные корректны
IF UB_0_32_AI8_UNITBUS_VAL_QUALITY_GROUP_1 = 3 AND
    UB_0_32_AI8_UNITBUS_VAL_QUALITY_GROUP_2 = 3

    THEN UB_0_32_AI8_UNITBUS_VAL_QUALITY := 3;
END_IF;

END_PROGRAM

(* ---- UB_local_0_38_AOC4.st ---- *)
PROGRAM UB_local_0_38_AOC4

(***************************************************************************)
// НАСТРОЙКА ФБ
(***************************************************************************)

UB_0_32_AOC4_CH0_VAL_QUALITY_AD.Valid_down := AD_VALID_DOWN;
UB_0_32_AOC4_CH0_VAL_QUALITY_AD.Valid_up := AD_VALID_UP;
UB_0_32_AOC4_CH0_VAL_QUALITY_AD.IN0 := AD_IN0;
UB_0_32_AOC4_CH0_VAL_QUALITY_AD.IN100 := AD_IN100;

UB_0_32_AOC4_CH0_VAL_DIAG_QUALITY_AD.Valid_down := AD_VALID_DOWN;
UB_0_32_AOC4_CH0_VAL_DIAG_QUALITY_AD.Valid_up := AD_VALID_UP;
UB_0_32_AOC4_CH0_VAL_DIAG_QUALITY_AD.IN0 := AD_IN0;
UB_0_32_AOC4_CH0_VAL_DIAG_QUALITY_AD.IN100 := AD_IN100;

UB_0_32_AOC4_CH1_VAL_QUALITY_AD.Valid_down := AD_VALID_DOWN;
UB_0_32_AOC4_CH1_VAL_QUALITY_AD.Valid_up := AD_VALID_UP;
UB_0_32_AOC4_CH1_VAL_QUALITY_AD.IN0 := AD_IN0;
UB_0_32_AOC4_CH1_VAL_QUALITY_AD.IN100 := AD_IN100;

UB_0_32_AOC4_CH1_VAL_DIAG_QUALITY_AD.Valid_down := AD_VALID_DOWN;
UB_0_32_AOC4_CH1_VAL_DIAG_QUALITY_AD.Valid_up := AD_VALID_UP;
UB_0_32_AOC4_CH1_VAL_DIAG_QUALITY_AD.IN0 := AD_IN0;
UB_0_32_AOC4_CH1_VAL_DIAG_QUALITY_AD.IN100 := AD_IN100;

UB_0_32_AOC4_CH2_VAL_QUALITY_AD.Valid_down := AD_VALID_DOWN;
UB_0_32_AOC4_CH2_VAL_QUALITY_AD.Valid_up := AD_VALID_UP;
UB_0_32_AOC4_CH2_VAL_QUALITY_AD.IN0 := AD_IN0;
UB_0_32_AOC4_CH2_VAL_QUALITY_AD.IN100 := AD_IN100;

UB_0_32_AOC4_CH2_VAL_DIAG_QUALITY_AD.Valid_down := AD_VALID_DOWN;
UB_0_32_AOC4_CH2_VAL_DIAG_QUALITY_AD.Valid_up := AD_VALID_UP;
UB_0_32_AOC4_CH2_VAL_DIAG_QUALITY_AD.IN0 := AD_IN0;
UB_0_32_AOC4_CH2_VAL_DIAG_QUALITY_AD.IN100 := AD_IN100;

UB_0_32_AOC4_CH3_VAL_QUALITY_AD.Valid_down := AD_VALID_DOWN;
UB_0_32_AOC4_CH3_VAL_QUALITY_AD.Valid_up := AD_VALID_UP;
UB_0_32_AOC4_CH3_VAL_QUALITY_AD.IN0 := AD_IN0;
UB_0_32_AOC4_CH3_VAL_QUALITY_AD.IN100 := AD_IN100;

UB_0_32_AOC4_CH3_VAL_DIAG_QUALITY_AD.Valid_down := AD_VALID_DOWN;
UB_0_32_AOC4_CH3_VAL_DIAG_QUALITY_AD.Valid_up := AD_VALID_UP;
UB_0_32_AOC4_CH3_VAL_DIAG_QUALITY_AD.IN0 := AD_IN0;
UB_0_32_AOC4_CH3_VAL_DIAG_QUALITY_AD.IN100 := AD_IN100;

(***************************************************************************)
// ЗАПИСЬ ЗНАЧЕНИЙ В КАНАЛЫ
(***************************************************************************)

_IO_Q23_AOC4_0_VAL.Measurement := ANY_TO_INT(REAL_TO_DINT(ABS(GENERATOR.Out_REAL), 0.0, 1500.0));
_IO_Q23_AOC4_1_VAL.Measurement := ANY_TO_INT(REAL_TO_DINT(ABS(GENERATOR.Out_REAL), 0.0, 1500.0));
_IO_Q23_AOC4_2_VAL.Measurement := ANY_TO_INT(REAL_TO_DINT(ABS(GENERATOR.Out_REAL), 0.0, 1500.0));
_IO_Q23_AOC4_3_VAL.Measurement := ANY_TO_INT(REAL_TO_DINT(ABS(GENERATOR.Out_REAL), 0.0, 1500.0));

(***************************************************************************)
// СБРОС ОШИБОК
(***************************************************************************)

IF UB_0_32_AOC4_KVIT
    THEN UB_0_32_AOC4_KVIT := FALSE;
END_IF;

(***************************************************************************)
// КАНАЛ 0
(***************************************************************************)

UB_0_32_AOC4_CH0_VAL_MEASUREMENT := _IO_Q23_AOC4_0_VAL.Measurement;
UB_0_32_AOC4_CH0_VAL_DIAG_MEASUREMENT := _IO_I23_AOC4_0_VAL_DIAG.Measurement;

//Отказ сигнала
IF INT14(ANY_TO_DINT(_IO_I23_AOC4_1_VAL_DIAG.Quality))
    THEN UB_0_32_AOC4_CH0_VAL_DIAG_QUALITY_FAULT := TRUE;
    ELSE UB_0_32_AOC4_CH0_VAL_DIAG_QUALITY_FAULT := FALSE;
END_IF;

// Проверка на ошибку
IF _IO_I23_AOC4_0_VAL_DIAG.Quality = 0
    THEN UB_0_32_AOC4_CH0_VAL_DIAG_QUALITY_ERROR := TRUE;
    ELSE UB_0_32_AOC4_CH0_VAL_DIAG_QUALITY_ERROR := FALSE;
END_IF;

(***************************************************************************)
// КАНАЛ 1
(***************************************************************************)

UB_0_32_AOC4_CH1_VAL_MEASUREMENT := _IO_Q23_AOC4_1_VAL.Measurement;
UB_0_32_AOC4_CH1_VAL_DIAG_MEASUREMENT := _IO_I23_AOC4_1_VAL_DIAG.Measurement;

//Отказ сигнала
IF INT14(ANY_TO_DINT(_IO_I23_AOC4_1_VAL_DIAG.Quality))
    THEN UB_0_32_AOC4_CH1_VAL_DIAG_QUALITY_FAULT := TRUE;
    ELSE UB_0_32_AOC4_CH1_VAL_DIAG_QUALITY_FAULT := FALSE;
END_IF;

// Проверка на ошибку
IF _IO_I23_AOC4_1_VAL_DIAG.Quality = 0
    THEN UB_0_32_AOC4_CH1_VAL_DIAG_QUALITY_ERROR := TRUE;
    ELSE UB_0_32_AOC4_CH1_VAL_DIAG_QUALITY_ERROR := FALSE;
END_IF;

(***************************************************************************)
// КАНАЛ 2
(***************************************************************************)

UB_0_32_AOC4_CH2_VAL_MEASUREMENT := _IO_Q23_AOC4_2_VAL.Measurement;
UB_0_32_AOC4_CH2_VAL_DIAG_MEASUREMENT := _IO_I23_AOC4_2_VAL_DIAG.Measurement;

//Отказ сигнала
IF INT14(ANY_TO_DINT(_IO_I23_AOC4_2_VAL_DIAG.Quality))
    THEN UB_0_32_AOC4_CH2_VAL_DIAG_QUALITY_FAULT := TRUE;
    ELSE UB_0_32_AOC4_CH2_VAL_DIAG_QUALITY_FAULT := FALSE;
END_IF;

// Проверка на ошибку
IF _IO_I23_AOC4_2_VAL_DIAG.Quality = 0
    THEN UB_0_32_AOC4_CH2_VAL_DIAG_QUALITY_ERROR := TRUE;
    ELSE UB_0_32_AOC4_CH2_VAL_DIAG_QUALITY_ERROR := FALSE;
END_IF;

(***************************************************************************)
// КАНАЛ 3
(***************************************************************************)

UB_0_32_AOC4_CH3_VAL_MEASUREMENT := _IO_Q23_AOC4_3_VAL.Measurement;
UB_0_32_AOC4_CH3_VAL_DIAG_MEASUREMENT := _IO_I23_AOC4_3_VAL_DIAG.Measurement;

//Отказ сигнала
IF INT14(ANY_TO_DINT(_IO_I23_AOC4_3_VAL_DIAG.Quality))
    THEN UB_0_32_AOC4_CH3_VAL_DIAG_QUALITY_FAULT := TRUE;
    ELSE UB_0_32_AOC4_CH3_VAL_DIAG_QUALITY_FAULT := FALSE;
END_IF;

// Проверка на ошибку
IF _IO_I23_AOC4_3_VAL_DIAG.Quality = 0
    THEN UB_0_32_AOC4_CH3_VAL_DIAG_QUALITY_ERROR := TRUE;
    ELSE UB_0_32_AOC4_CH3_VAL_DIAG_QUALITY_ERROR := FALSE;
END_IF;

(***************************************************************************)
// ИНТЕГРАЛЬНЫЕ ПОКАЗАТЕЛИ
(***************************************************************************)

// Интегральный показателшь VAL.Quality
IF NOT INT0(UB_0_32_AOC4_CH0_VAL_QUALITY) AND
    NOT INT0(UB_0_32_AOC4_CH1_VAL_QUALITY) AND
    NOT INT0(UB_0_32_AOC4_CH2_VAL_QUALITY) AND
    NOT INT0(UB_0_32_AOC4_CH3_VAL_QUALITY)

    THEN UB_0_32_AOC4_INTEGRAL_VAL_QUALITY := TRUE;
    ELSE UB_0_32_AOC4_INTEGRAL_VAL_QUALITY := FALSE;
END_IF;

// Интегральный показателшь VAL_DIAG.Quality
IF NOT INT0(UB_0_32_AOC4_CH0_VAL_DIAG_QUALITY) AND
    NOT INT0(UB_0_32_AOC4_CH1_VAL_DIAG_QUALITY) AND
    NOT INT0(UB_0_32_AOC4_CH2_VAL_DIAG_QUALITY) AND
    NOT INT0(UB_0_32_AOC4_CH3_VAL_DIAG_QUALITY)

    THEN UB_0_32_AOC4_INTEGRAL_VAL_DIAG_QUALITY := TRUE;
    ELSE UB_0_32_AOC4_INTEGRAL_VAL_DIAG_QUALITY := FALSE;
END_IF;

(***************************************************************************)
// ДИАГНОСТИКА ШИНЫ
(***************************************************************************)

// VAL.Quality
// Адресное пространство не было найдено в Ubusdb
IF
    // Канал 0
    NOT INT4(ANY_TO_DINT(_IO_Q23_AOC4_0_VAL.Quality)) AND
    NOT INT5(ANY_TO_DINT(_IO_Q23_AOC4_0_VAL.Quality)) AND
    NOT INT6(ANY_TO_DINT(_IO_Q23_AOC4_0_VAL.Quality)) AND
    NOT INT7(ANY_TO_DINT(_IO_Q23_AOC4_0_VAL.Quality)) AND

    // Канал 1
    NOT INT4(ANY_TO_DINT(_IO_Q23_AOC4_1_VAL.Quality)) AND
    NOT INT5(ANY_TO_DINT(_IO_Q23_AOC4_1_VAL.Quality)) AND
    NOT INT6(ANY_TO_DINT(_IO_Q23_AOC4_1_VAL.Quality)) AND
    NOT INT7(ANY_TO_DINT(_IO_Q23_AOC4_1_VAL.Quality)) AND

    // Канал 2
    NOT INT4(ANY_TO_DINT(_IO_Q23_AOC4_2_VAL.Quality)) AND
    NOT INT5(ANY_TO_DINT(_IO_Q23_AOC4_2_VAL.Quality)) AND
    NOT INT6(ANY_TO_DINT(_IO_Q23_AOC4_2_VAL.Quality)) AND
    NOT INT7(ANY_TO_DINT(_IO_Q23_AOC4_2_VAL.Quality)) AND

    // Канал 3
    NOT INT4(ANY_TO_DINT(_IO_Q23_AOC4_3_VAL.Quality)) AND
    NOT INT5(ANY_TO_DINT(_IO_Q23_AOC4_3_VAL.Quality)) AND
    NOT INT6(ANY_TO_DINT(_IO_Q23_AOC4_3_VAL.Quality)) AND
    NOT INT7(ANY_TO_DINT(_IO_Q23_AOC4_3_VAL.Quality))

    THEN UB_0_32_AOC4_UNITBUS_VAL_QUALITY := 0;
END_IF;

// Не сошлась контрольная сумма данных
IF
    // Канал 0
    INT4(ANY_TO_DINT(_IO_Q23_AOC4_0_VAL.Quality)) AND
    NOT INT5(ANY_TO_DINT(_IO_Q23_AOC4_0_VAL.Quality)) AND
    NOT INT6(ANY_TO_DINT(_IO_Q23_AOC4_0_VAL.Quality)) AND
    NOT INT7(ANY_TO_DINT(_IO_Q23_AOC4_0_VAL.Quality)) AND

    // Канал 1
    INT4(ANY_TO_DINT(_IO_Q23_AOC4_1_VAL.Quality)) AND
    NOT INT5(ANY_TO_DINT(_IO_Q23_AOC4_1_VAL.Quality)) AND
    NOT INT6(ANY_TO_DINT(_IO_Q23_AOC4_1_VAL.Quality)) AND
    NOT INT7(ANY_TO_DINT(_IO_Q23_AOC4_1_VAL.Quality)) AND

    // Канал 2
    INT4(ANY_TO_DINT(_IO_Q23_AOC4_2_VAL.Quality)) AND
    NOT INT5(ANY_TO_DINT(_IO_Q23_AOC4_2_VAL.Quality)) AND
    NOT INT6(ANY_TO_DINT(_IO_Q23_AOC4_2_VAL.Quality)) AND
    NOT INT7(ANY_TO_DINT(_IO_Q23_AOC4_2_VAL.Quality)) AND

    // Канал 3
    INT4(ANY_TO_DINT(_IO_Q23_AOC4_3_VAL.Quality)) AND
    NOT INT5(ANY_TO_DINT(_IO_Q23_AOC4_3_VAL.Quality)) AND
    NOT INT6(ANY_TO_DINT(_IO_Q23_AOC4_3_VAL.Quality)) AND
    NOT INT7(ANY_TO_DINT(_IO_Q23_AOC4_3_VAL.Quality))

    THEN UB_0_32_AOC4_UNITBUS_VAL_QUALITY := 1;
END_IF;

// Не выставлены биты достоверности элементов в АП
IF
    // Канал 0
    NOT INT4(ANY_TO_DINT(_IO_Q23_AOC4_0_VAL.Quality)) AND
    INT5(ANY_TO_DINT(_IO_Q23_AOC4_0_VAL.Quality)) AND
    NOT INT6(ANY_TO_DINT(_IO_Q23_AOC4_0_VAL.Quality)) AND
    NOT INT7(ANY_TO_DINT(_IO_Q23_AOC4_0_VAL.Quality)) AND

    // Канал 1
    NOT INT4(ANY_TO_DINT(_IO_Q23_AOC4_1_VAL.Quality)) AND
    INT5(ANY_TO_DINT(_IO_Q23_AOC4_1_VAL.Quality)) AND
    NOT INT6(ANY_TO_DINT(_IO_Q23_AOC4_1_VAL.Quality)) AND
    NOT INT7(ANY_TO_DINT(_IO_Q23_AOC4_1_VAL.Quality)) AND

    // Канал 2
    NOT INT4(ANY_TO_DINT(_IO_Q23_AOC4_2_VAL.Quality)) AND
    INT5(ANY_TO_DINT(_IO_Q23_AOC4_2_VAL.Quality)) AND
    NOT INT6(ANY_TO_DINT(_IO_Q23_AOC4_2_VAL.Quality)) AND
    NOT INT7(ANY_TO_DINT(_IO_Q23_AOC4_2_VAL.Quality)) AND

    // Канал 3
    NOT INT4(ANY_TO_DINT(_IO_Q23_AOC4_3_VAL.Quality)) AND
    INT5(ANY_TO_DINT(_IO_Q23_AOC4_3_VAL.Quality)) AND
    NOT INT6(ANY_TO_DINT(_IO_Q23_AOC4_3_VAL.Quality)) AND
    NOT INT7(ANY_TO_DINT(_IO_Q23_AOC4_3_VAL.Quality))

    THEN UB_0_32_AOC4_UNITBUS_VAL_QUALITY := 2;
END_IF;

// Полученные данные корректны
IF
    // Канал 0
    INT4(ANY_TO_DINT(_IO_Q23_AOC4_0_VAL.Quality)) AND
    INT5(ANY_TO_DINT(_IO_Q23_AOC4_0_VAL.Quality)) AND
    NOT INT6(ANY_TO_DINT(_IO_Q23_AOC4_0_VAL.Quality)) AND
    NOT INT7(ANY_TO_DINT(_IO_Q23_AOC4_0_VAL.Quality)) AND

    // Канал 1
    INT4(ANY_TO_DINT(_IO_Q23_AOC4_1_VAL.Quality)) AND
    INT5(ANY_TO_DINT(_IO_Q23_AOC4_1_VAL.Quality)) AND
    NOT INT6(ANY_TO_DINT(_IO_Q23_AOC4_1_VAL.Quality)) AND
    NOT INT7(ANY_TO_DINT(_IO_Q23_AOC4_1_VAL.Quality)) AND

    // Канал 2
    INT4(ANY_TO_DINT(_IO_Q23_AOC4_2_VAL.Quality)) AND
    INT5(ANY_TO_DINT(_IO_Q23_AOC4_2_VAL.Quality)) AND
    NOT INT6(ANY_TO_DINT(_IO_Q23_AOC4_2_VAL.Quality)) AND
    NOT INT7(ANY_TO_DINT(_IO_Q23_AOC4_2_VAL.Quality)) AND

    // Канал 3
    INT4(ANY_TO_DINT(_IO_Q23_AOC4_3_VAL.Quality)) AND
    INT5(ANY_TO_DINT(_IO_Q23_AOC4_3_VAL.Quality)) AND
    NOT INT6(ANY_TO_DINT(_IO_Q23_AOC4_3_VAL.Quality)) AND
    NOT INT7(ANY_TO_DINT(_IO_Q23_AOC4_3_VAL.Quality))

    THEN UB_0_32_AOC4_UNITBUS_VAL_QUALITY := 3;
END_IF;

// VAL_DIAG.Quality
// Адресное пространство не было найдено в Ubusdb
IF
    // Канал 0
    NOT INT4(ANY_TO_DINT(_IO_I23_AOC4_0_VAL_DIAG.Quality)) AND
    NOT INT5(ANY_TO_DINT(_IO_I23_AOC4_0_VAL_DIAG.Quality)) AND
    NOT INT6(ANY_TO_DINT(_IO_I23_AOC4_0_VAL_DIAG.Quality)) AND
    NOT INT7(ANY_TO_DINT(_IO_I23_AOC4_0_VAL_DIAG.Quality)) AND

    // Канал 1
    NOT INT4(ANY_TO_DINT(_IO_I23_AOC4_1_VAL_DIAG.Quality)) AND
    NOT INT5(ANY_TO_DINT(_IO_I23_AOC4_1_VAL_DIAG.Quality)) AND
    NOT INT6(ANY_TO_DINT(_IO_I23_AOC4_1_VAL_DIAG.Quality)) AND
    NOT INT7(ANY_TO_DINT(_IO_I23_AOC4_1_VAL_DIAG.Quality)) AND

    // Канал 2
    NOT INT4(ANY_TO_DINT(_IO_I23_AOC4_2_VAL_DIAG.Quality)) AND
    NOT INT5(ANY_TO_DINT(_IO_I23_AOC4_2_VAL_DIAG.Quality)) AND
    NOT INT6(ANY_TO_DINT(_IO_I23_AOC4_2_VAL_DIAG.Quality)) AND
    NOT INT7(ANY_TO_DINT(_IO_I23_AOC4_2_VAL_DIAG.Quality)) AND

    // Канал 3
    NOT INT4(ANY_TO_DINT(_IO_I23_AOC4_3_VAL_DIAG.Quality)) AND
    NOT INT5(ANY_TO_DINT(_IO_I23_AOC4_3_VAL_DIAG.Quality)) AND
    NOT INT6(ANY_TO_DINT(_IO_I23_AOC4_3_VAL_DIAG.Quality)) AND
    NOT INT7(ANY_TO_DINT(_IO_I23_AOC4_3_VAL_DIAG.Quality))

    THEN UB_0_32_AOC4_UNITBUS_VAL_DIAG_QUALITY := 0;
END_IF;

// Не сошлась контрольная сумма данных
IF
    // Канал 0
    INT4(ANY_TO_DINT(_IO_I23_AOC4_0_VAL_DIAG.Quality)) AND
    NOT INT5(ANY_TO_DINT(_IO_I23_AOC4_0_VAL_DIAG.Quality)) AND
    NOT INT6(ANY_TO_DINT(_IO_I23_AOC4_0_VAL_DIAG.Quality)) AND
    NOT INT7(ANY_TO_DINT(_IO_I23_AOC4_0_VAL_DIAG.Quality)) AND

    // Канал 1
    INT4(ANY_TO_DINT(_IO_I23_AOC4_1_VAL_DIAG.Quality)) AND
    NOT INT5(ANY_TO_DINT(_IO_I23_AOC4_1_VAL_DIAG.Quality)) AND
    NOT INT6(ANY_TO_DINT(_IO_I23_AOC4_1_VAL_DIAG.Quality)) AND
    NOT INT7(ANY_TO_DINT(_IO_I23_AOC4_1_VAL_DIAG.Quality)) AND

    // Канал 2
    INT4(ANY_TO_DINT(_IO_I23_AOC4_2_VAL_DIAG.Quality)) AND
    NOT INT5(ANY_TO_DINT(_IO_I23_AOC4_2_VAL_DIAG.Quality)) AND
    NOT INT6(ANY_TO_DINT(_IO_I23_AOC4_2_VAL_DIAG.Quality)) AND
    NOT INT7(ANY_TO_DINT(_IO_I23_AOC4_2_VAL_DIAG.Quality)) AND

    // Канал 3
    INT4(ANY_TO_DINT(_IO_I23_AOC4_3_VAL_DIAG.Quality)) AND
    NOT INT5(ANY_TO_DINT(_IO_I23_AOC4_3_VAL_DIAG.Quality)) AND
    NOT INT6(ANY_TO_DINT(_IO_I23_AOC4_3_VAL_DIAG.Quality)) AND
    NOT INT7(ANY_TO_DINT(_IO_I23_AOC4_3_VAL_DIAG.Quality))

    THEN UB_0_32_AOC4_UNITBUS_VAL_DIAG_QUALITY := 1;
END_IF;

// Не выставлены биты достоверности элементов в АП
IF
    // Канал 0
    NOT INT4(ANY_TO_DINT(_IO_I23_AOC4_0_VAL_DIAG.Quality)) AND
    INT5(ANY_TO_DINT(_IO_I23_AOC4_0_VAL_DIAG.Quality)) AND
    NOT INT6(ANY_TO_DINT(_IO_I23_AOC4_0_VAL_DIAG.Quality)) AND
    NOT INT7(ANY_TO_DINT(_IO_I23_AOC4_0_VAL_DIAG.Quality)) AND

    // Канал 1
    NOT INT4(ANY_TO_DINT(_IO_I23_AOC4_1_VAL_DIAG.Quality)) AND
    INT5(ANY_TO_DINT(_IO_I23_AOC4_1_VAL_DIAG.Quality)) AND
    NOT INT6(ANY_TO_DINT(_IO_I23_AOC4_1_VAL_DIAG.Quality)) AND
    NOT INT7(ANY_TO_DINT(_IO_I23_AOC4_1_VAL_DIAG.Quality)) AND

    // Канал 2
    NOT INT4(ANY_TO_DINT(_IO_I23_AOC4_2_VAL_DIAG.Quality)) AND
    INT5(ANY_TO_DINT(_IO_I23_AOC4_2_VAL_DIAG.Quality)) AND
    NOT INT6(ANY_TO_DINT(_IO_I23_AOC4_2_VAL_DIAG.Quality)) AND
    NOT INT7(ANY_TO_DINT(_IO_I23_AOC4_2_VAL_DIAG.Quality)) AND

    // Канал 3
    NOT INT4(ANY_TO_DINT(_IO_I23_AOC4_3_VAL_DIAG.Quality)) AND
    INT5(ANY_TO_DINT(_IO_I23_AOC4_3_VAL_DIAG.Quality)) AND
    NOT INT6(ANY_TO_DINT(_IO_I23_AOC4_3_VAL_DIAG.Quality)) AND
    NOT INT7(ANY_TO_DINT(_IO_I23_AOC4_3_VAL_DIAG.Quality))

    THEN UB_0_32_AOC4_UNITBUS_VAL_DIAG_QUALITY := 2;
END_IF;

// Полученные данные корректны
IF
    // Канал 0
    INT4(ANY_TO_DINT(_IO_I23_AOC4_0_VAL_DIAG.Quality)) AND
    INT5(ANY_TO_DINT(_IO_I23_AOC4_0_VAL_DIAG.Quality)) AND
    NOT INT6(ANY_TO_DINT(_IO_I23_AOC4_0_VAL_DIAG.Quality)) AND
    NOT INT7(ANY_TO_DINT(_IO_I23_AOC4_0_VAL_DIAG.Quality)) AND

    // Канал 1
    INT4(ANY_TO_DINT(_IO_I23_AOC4_1_VAL_DIAG.Quality)) AND
    INT5(ANY_TO_DINT(_IO_I23_AOC4_1_VAL_DIAG.Quality)) AND
    NOT INT6(ANY_TO_DINT(_IO_I23_AOC4_1_VAL_DIAG.Quality)) AND
    NOT INT7(ANY_TO_DINT(_IO_I23_AOC4_1_VAL_DIAG.Quality)) AND

    // Канал 2
    INT4(ANY_TO_DINT(_IO_I23_AOC4_2_VAL_DIAG.Quality)) AND
    INT5(ANY_TO_DINT(_IO_I23_AOC4_2_VAL_DIAG.Quality)) AND
    NOT INT6(ANY_TO_DINT(_IO_I23_AOC4_2_VAL_DIAG.Quality)) AND
    NOT INT7(ANY_TO_DINT(_IO_I23_AOC4_2_VAL_DIAG.Quality)) AND

    // Канал 3
    INT4(ANY_TO_DINT(_IO_I23_AOC4_3_VAL_DIAG.Quality)) AND
    INT5(ANY_TO_DINT(_IO_I23_AOC4_3_VAL_DIAG.Quality)) AND
    NOT INT6(ANY_TO_DINT(_IO_I23_AOC4_3_VAL_DIAG.Quality)) AND
    NOT INT7(ANY_TO_DINT(_IO_I23_AOC4_3_VAL_DIAG.Quality))

    THEN UB_0_32_AOC4_UNITBUS_VAL_DIAG_QUALITY := 3;
END_IF;

END_PROGRAM
